FUNCTION_BLOCK TEST_SEL2 (* Test Misc SEL functions *)
  (* Standard: IEC 61499-1 *)
  (* Version 0.0, 2006-09-14, JHC, Holobloc Inc *)
  (* Compiler header: package fb.rt.test; *)
  (* Compiler classdef: SimpleFB *)
  (* Compiler Java Sun JDK 1.5.0 *)
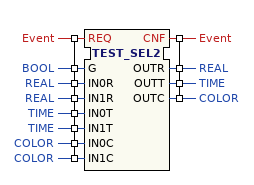
  EVENT_INPUT
    REQ WITH IN1R, IN0R, IN0T, G, IN1T, IN0C, IN1C;
  END_EVENT
  EVENT_OUTPUT
    CNF WITH OUTR, OUTT, OUTC;
  END_EVENT
  VAR_INPUT
    G : BOOL; (* Selection gate *)
    IN0R : REAL;
    IN1R : REAL;
    IN0T : TIME;
    IN1T : TIME;
    IN0C : COLOR;
    IN1C : COLOR;
  END_VAR
  VAR_OUTPUT
    OUTR : REAL;
    OUTT : TIME;
    OUTC : COLOR;
  END_VAR
  ALGORITHM REQ IN FBD:
    FBS
      SELR : SEL_REAL;
      SELT : SEL_TIME;
      SELC : SEL_COLOR;
    END_FBS
    DATA_CONNECTIONS
      IN1R TO SELR.IN1;
      SELR.OUT TO OUTR;
      IN1T TO SELT.IN1;
      SELT.OUT TO OUTT;
      G TO SELR.G;
      IN0R TO SELR.IN0;
      G TO SELT.G;
      IN0T TO SELT.IN0;
      G TO SELC.G;
      IN0C TO SELC.IN0;
      IN1C TO SELC.IN1;
      SELC.OUT TO OUTC;
    END_CONNECTIONS
  END_ALGORITHM
END_FUNCTION_BLOCK
